(* IEC 61131-3 sources: YaoKangDeviceDemo/src/30_Task, 2 files *)

(* ---- PRG_ParamService.st ---- *)
(*============================================================================
  PRG_ParamService —— 层 30 任务：参数管理服务（扫描链第 8 环）
  ----------------------------------------------------------------------------
  唯一写入：内部参数运行区/编辑缓冲/Retain（P5 建内部模型结构体）；
            各 ConfigCmd 的 bSuccess/bError/iErrorCode 回令；身份块
            HMI_DeviceIdentity / HMI_DeviceIdentityWrite。
  读入：  HMI.*.ConfigCmd（bLoad/bApply/bSave/bResetDefault）、
          HMI_DeviceIdentityWrite.Cmd（身份块仅 bLoad/bApply）。
  三区模型：运行区（生效）/ 编辑缓冲（HMI 线上编辑区）/ Retain（断电保持）。
  P1：骨架。
  P5：FC_ValidateParams 校验拒绝（返回 iParamError+轴+字段三元组）、
      工厂默认、运行中锁存快照、Retain（含 bZeroCommissioned）。
  P11：设备身份 Load/Apply，非法/锁定报 5005/5006；D1000 镜像 + MAC 回填。
==========================================================================*)
PROGRAM PRG_ParamService
VAR
END_VAR

(* TODO P5: 统一处理 5 个 Stru_ConfigCmd 实例：
     HMI.Condition.ParamCmd / HMI.TailTilt.ConfigCmd /
     HMI.ChestImpact.ConfigCmd / HMI.SeatTwist.ConfigCmd /
     HMI.LegAngle.ConfigCmd / HMI.HomingParams.Cmd
   脉冲位由 INPUT_ADAPTER 的 R_TRIG 解析后（P2 补 trig），按：
     bLoad   : 运行区 → 编辑缓冲（HMI 线上区）
     bApply  : 编辑缓冲 → FC_ValidateParams 校验 → 通过则覆盖运行区，失败回 iErrorCode
     bSave   : 运行区 → Retain
     bResetDefault : 工厂默认 → 运行区/缓冲
   回令：成功置 bSuccess、失败置 bError+iErrorCode，命令位由 InputAdapter 回清。 *)

(* TODO P11: 设备身份（D1000–D1013）
   - 每扫回填只读镜像 HMI_DeviceIdentity：
       diDeviceNoRaw := Retain 设备编号；
       iMacWord0/1/2 := _Ethernet.MACAddress[0..2]（H5U 系统变量，P11 核对名称）。
   - HMI_DeviceIdentityWrite.Cmd：bLoad 回读当前编号；bApply 校验+权限/锁定
     判定后写入 Retain，失败回 bError + 5005（锁定）/5006（非法）。 *)
END_PROGRAM

(* ---- PRG_TaskRunner.st ---- *)
(*============================================================================
  PRG_TaskRunner —— 层 30 任务：任务调度（扫描链第 7 环）
  ----------------------------------------------------------------------------
  唯一写入：iPhase（任务内阶段上报）、iBlockReason（阻塞原因）；任务级
            Cmd/Motion（HMI 各轴/推杆 Cmd 与 Motion 参数块）；故障经 gFaultSubmit。
  读入：  iState（MODE_MANAGER）、trig* 命令边沿、内部运行区参数。
  分派：按 iState 调度 AUTORUN（FBI_Cond/FATIGUE）/SELFTEST/HOMING/
        CALIBRATE/RESET 任务；任务模块只写任务级命令，MC 指令由
        OUTPUT_ADAPTER 唯一执行；不直接切 iState。
  P1：状态分派占位。
  P9/P10：回零/紧急回零/自检/建零、调理/治疗/老化自动流程。
==========================================================================*)
PROGRAM PRG_TaskRunner
VAR
END_VAR

CASE iState OF
    ST_STANDBY:
        (* TODO P6/P10: 就绪态等待启动；快速启动/自动流程入口门控 *)
        iPhase := COND_IDLE;

    ST_AUTORUN:
        (* TODO P10: FBI_Cond（调理/治疗）/ FATIGUE（老化）状态机
           105 启动前检查 → 108 等待准备 → 110 成角 → 120 等确认
           → 130 三轴 16 段联动 → 140 安全降落 → 800 完成 / 900 异常 *)
        ;

    ST_SELFTEST:
        (* TODO P9: 动态自检 Step10→100/200（推杆参考检查→成角→三轴 ±2°→回零） *)
        ;

    ST_HOMING:
        (* TODO P9: 普通回零（三轴 MoveAbs 回初始位）；紧急回零在 SOFT_ESTOP 内 *)
        ;

    ST_CALIBRATE:
        (* TODO P8/P9: 推杆校准 / 维护建零（6 重门控后 MC_Home/标定） *)
        ;

    ST_RESET:
        (* TODO P9: 故障复位收口：清错误、回初始位、完成后回 STANDBY（由 ModeManager 切） *)
        iPhase := 0;
        iState := ST_STANDBY;   (* TODO: 复位流程完成后再切，P6 收口仲裁时移回 ModeManager *)

    ST_STOPPING, ST_SOFT_ESTOP, ST_HARD_ESTOP:
        (* 安全收口由 SAFETY_MANAGER / POWER / OUTPUT_ADAPTER 执行，任务层不动作 *)
        ;
ELSE
    (* INIT / READY_CHECK / SERVICE / SERVICE_REQUIRED / PARAM_LIMITED：P6/P11 补 *)
    ;
END_CASE;
END_PROGRAM
